# EPICS autosave request: asApp/Db/configMenuNames.req
$(P)$(CONFIG)Menu:name1
$(P)$(CONFIG)Menu:name2
$(P)$(CONFIG)Menu:name3
$(P)$(CONFIG)Menu:name4
$(P)$(CONFIG)Menu:name5
$(P)$(CONFIG)Menu:name6
$(P)$(CONFIG)Menu:name7
$(P)$(CONFIG)Menu:name8
$(P)$(CONFIG)Menu:name9
$(P)$(CONFIG)Menu:name10
$(P)$(CONFIG)Menu:desc1
$(P)$(CONFIG)Menu:desc2
$(P)$(CONFIG)Menu:desc3
$(P)$(CONFIG)Menu:desc4
$(P)$(CONFIG)Menu:desc5
$(P)$(CONFIG)Menu:desc6
$(P)$(CONFIG)Menu:desc7
$(P)$(CONFIG)Menu:desc8
$(P)$(CONFIG)Menu:desc9
$(P)$(CONFIG)Menu:desc10
